# EPICS substitutions: iocBoot/ioc13bmc/auto_shutter.substitutions
file "$(CARS)/CARSApp/Db/auto_shutter_old.db"
{
pattern
{P,      SHUT,      SHUT_STATUS,         SHUT_CONTROL}
{13BMC:, BMC,     13BMA:eps_mbbi100,     13BMA:OpenBMCShutter}
}
